DATA_BLOCK "OPC_DB"
{ S7_Optimized_Access := 'TRUE' }
VERSION : 0.1
NON_RETAIN
   VAR RETAIN
      X : Real;
      Y : Real;
   END_VAR


BEGIN

END_DATA_BLOCK

